// TIA Portal V19 export
VAR_GLOBAL   // PLC tag table "CC1"
   CC1_HighTemperature AT %I0.6 : Bool;   // 110S2 - Temperatura > 45°C
   CC1_ThermalTrip24Vdc_PLC_SINAMICS AT %I1.7 : Bool;   // 133QF1 - 24Vdc thermal trip PLC & SINAMICS
   CC1_ThermalTrip24Vdc_Valves AT %I100.4 : Bool;   // 135QF1 - 24Vdc thermal trip valves
   ThermalProtection_220V_Socket AT %I0.3 : Bool;   // 105QF1 - Thermal trip circuit 220v for service sockets
   CC1_Apertura_Porte AT %I0.0 : Bool;   // 102KA2
   PAC_Multifunzione_1 AT %Q0.0 : Bool;   // 103KA1 - NON USATO
   PAC_Multifunzione_2 AT %Q0.1 : Bool;   // 103KA2 - NON USATO
   PAC_7KM_1 AT %I0.1 : Bool;   // 103KA1 NON USATO
   PAC_7KM_2 AT %I0.2 : Bool;   // 103KA2 NON USATO
   CC1_Guasto_Condizionatore_1 AT %I0.4 : Bool;   // 110 -- 1= OK 0= FAULT
   CC1_Controllo_Temperatura_Quadro AT %I0.5 : Bool;   // 110S1 - Temperatura > 30°C
   CC1_Controllo_Circuito_Raffredamento_Quadro_1 AT %I0.7 : Bool;   // 110QF1
   CC1_ON_Condizionatori AT %Q0.2 : Bool;   // 110KM1
   CC1_Guasto_Condizionatore_2 AT %I1.0 : Bool;   // 112 -- 1= OK 0= FAULT
   CC1_Controllo_Circuito_Raffredamento_Quadro_2 AT %I1.1 : Bool;   // 112QF1
   JB001_ON_Condizionatore AT %Q100.0 : Bool;   // 109KA2
   JB001_Controllo_Temperatura_Quadro AT %I100.1 : Bool;   // 114S1 - Temperatura > 30°C
   JB001_Max_Temperatura_Quadro AT %I100.2 : Bool;   // 114S2 - Temperatura > 45°C
   JB001_Controllo_Circuito_Raffredamento_Quadro AT %I100.3 : Bool;   // 114QF1
   "24V_Batteria_Scarica" AT %I1.2 : Bool;   // 121 - SITOP UPS500S
   "24V_Allarme_Batteria" AT %I1.3 : Bool;   // 121 - SITOP UPS500S
   "24V_Batteria_OK" AT %I1.4 : Bool;   // 121 - SITOP UPS500S
   CC1_Ai_GeneralPressure_Air AT %IW904 : Int;   // 464A1 - 774B3
   "24V_Fdbk_Protezione_Elettronica" AT %I1.5 : Bool;   // 126 - SITOP SEL1400
   "24V_Controllo_Magnetotermico_Sinamics" AT %I1.6 : Bool;   // 132QF1
   CC1_Pressione_Aria_Generale_OK AT %I102.5 : Bool;   // 174S1
   Area01_Aspo_Pressione_Aria_OK AT %I102.6 : Bool;   // 176S1
   "24V_Reset_Protezione_Elettronica" AT %Q0.3 : Bool;   // 126 - SITOP SEL1400
   Scalance_XC216_Switch_ON AT %I2.5 : Bool;   // 392A1
   Scalance_XC116_1_Switch_ON AT %I2.6 : Bool;   // 394A1
   Scalance_XC116_2_Switch_ON AT %I2.7 : Bool;   // 396A1
   "Scalance_SC632-2C_Switch_ON" AT %I3.0 : Bool;   // 398A1
   CU320_Trigger_Lettura_Correzione_Encoder AT %Q0.4 : Bool;   // 588 - CU320
   CU320_Trigger_Lettrua_Taglio AT %Q0.5 : Bool;   // 588 - CU320
   Area02_03_Accoppiamento_Pressione_Aria_OK AT %I205.1 : Bool;   // 180S1
   Area03_Pareggiamneto_Pressione_Aria_OK AT %I300.2 : Bool;   // 182S1
   Area04_Navetta_Pressione_Aria_OK AT %I310.0 : Bool;   // 183S1
END_VAR
